FUNCTION TryConvert_UINT_TO_TOD : BOOL
VAR_INPUT
	in : UINT;
	out : REFERENCE TO TOD;
END_VAR

out := UINT_TO_TOD(in);
TryConvert_UINT_TO_TOD := TRUE;

END_FUNCTION

(* stored: Version 1.1.0.1, ProductVersion 3.1.4024.12
   POU TryConvert_UINT_TO_TOD: Id {3c768c42-81ac-40a7-8be2-0eb9a35d6e46}, SpecialFunc None *)
